// TIA Portal project "Tetsi" (V15.1)

(* hardware
DEVICE "S71500/ET200MP station_1"  S7-1500 station
   slot 0: "Rail_0"  Rack  6ES7 590-1***0-0AA0
   slot 1: "PLC_1"  CPU 1511-1 PN  6ES7 511-1AK02-0AB0  V2.6
      slot 3: "CPU display_1"  6ES7591-1AA00-0AA0
   slot 2: "DI 16x24VDC / DQ 16x24VDC/0.5A BA_1"  DI 16/DQ 16x24VDC  6ES7 523-1BL00-0AA0  V1.0
   slot 3: "AI/AQ 4xU/I/RTD/TC / 2xU/I ST_1"  AI/AQ 4xU/I/RTD/TC / 2xU/I ST  6ES7 534-7QE00-0AB0  V1.0
*)

// ===== PLC "PLC_1"  CPU 1511-1 PN =====

VAR_GLOBAL   // PLC tag table "Default tag table"
   "Clock_Byte" AT %MB0 : Byte;
   "Clock_10Hz" AT %M0.0 : Bool;
   "Clock_5Hz" AT %M0.1 : Bool;
   "Clock_2.5Hz" AT %M0.2 : Bool;
   "Clock_2Hz" AT %M0.3 : Bool;
   "Clock_1.25Hz" AT %M0.4 : Bool;
   "Clock_1Hz" AT %M0.5 : Bool;
   "Clock_0.625Hz" AT %M0.6 : Bool;
   "Clock_0.5Hz" AT %M0.7 : Bool;
   "Tag_1" AT %M10.0 : Bool;
   "kayntivalmius" AT %M10.1 : Bool;
END_VAR

VAR_GLOBAL   // PLC tag table "Tagit"
   "start" AT %I0.0 : Bool;
   "stop" AT %I0.1 : Bool;
   "anturi1" AT %I0.2 : Bool;
   "anturi2" AT %I0.3 : Bool;
   "turvakytkin" AT %I0.4 : Bool;
   "moottori1" AT %Q0.0 : Bool;
   "moottori2" AT %Q0.1 : Bool;
END_VAR

DATA_BLOCK "DB"   // DB1
{ S7_Optimized_Access := 'FALSE' }
VERSION : 0.1
   VAR
      nLaatikoita : Int;
   END_VAR
BEGIN
END_DATA_BLOCK

DATA_BLOCK "Data_block_1"   // DB2
{ S7_Optimized_Access := 'FALSE' }
VERSION : 0.1
   VAR
      start : Bool;
      stop : Bool;
      anturi1 : Bool;
      turvakytkin : Bool;
      moottori1 : Bool;
   END_VAR
BEGIN
END_DATA_BLOCK

ORGANIZATION_BLOCK "Main"   // OB1, LAD, ProgramCycle
TITLE = "Main Program Sweep (Cycle)"
{ S7_Optimized_Access := 'TRUE' }
VERSION : 0.1
   VAR_INPUT
      Initial_Call : Bool;   // Initial call of this OB
      Remanence : Bool;   // =True, if remanent data are available
   END_VAR
   VAR_TEMP   // added for the SCL form of the ladder/FBD networks
      _w1 : Bool;
   END_VAR
BEGIN

REGION Network 1
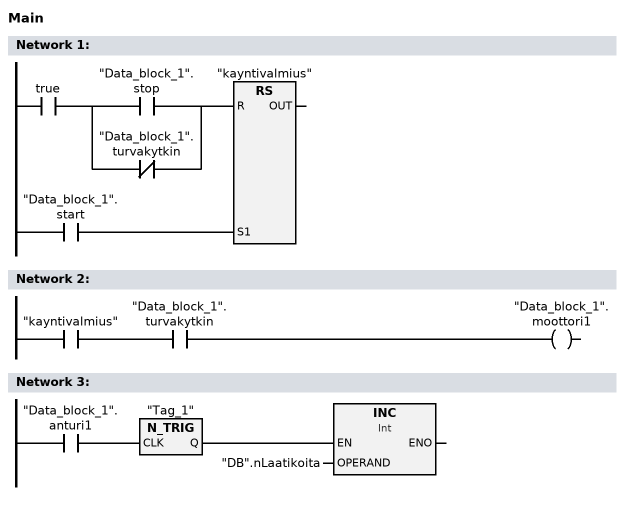
   RUNG wire#powerrail
      Contact( true )
      wire#w1
      Contact( "Data_block_1".stop )
      wire#w2
      S_RS(operand := "kayntivalmius", s1 := wire#w3)
   END_RUNG
   RUNG wire#w1
      I_Contact( "Data_block_1".turvakytkin )
   END_RUNG wire#w2
   RUNG wire#powerrail
      Contact( "Data_block_1".start )
   END_RUNG wire#w3
   // the same network as SCL:
   IF true AND ("Data_block_1".stop OR NOT "Data_block_1".turvakytkin) THEN
       "kayntivalmius" := FALSE;   // RS flip-flop
   END_IF;
   IF "Data_block_1".start THEN "kayntivalmius" := TRUE; END_IF;
END_REGION

REGION Network 2
   RUNG wire#powerrail
      Contact( "kayntivalmius" )
      Contact( "Data_block_1".turvakytkin )
      Coil( "Data_block_1".moottori1 )
   END_RUNG
   // the same network as SCL:
   "Data_block_1".moottori1 := "kayntivalmius" AND "Data_block_1".turvakytkin;
END_REGION

REGION Network 3
   RUNG wire#powerrail
      Contact( "Data_block_1".anturi1 )
      N_Trig( "Tag_1" )
      { S7_Templates := "DestType := Int" } Inc( "DB".nLaatikoita )
   END_RUNG
   // the same network as SCL:
   #_w1 := NOT "Data_block_1".anturi1 AND "Tag_1";   // falling edge
   "Tag_1" := "Data_block_1".anturi1;
   IF #_w1 THEN "DB".nLaatikoita := "DB".nLaatikoita + 1; END_IF;
END_REGION
END_ORGANIZATION_BLOCK